Universal Robots PolyScope program: prod_v5.urp

Program prod_v5 (installation=prod directory=/home/ur/ursim-current/programs/programs.UR10 createdIn=3.14.1.1031110 lastSavedIn=3.14.1.1031110 robotSerialNumber=2018309999)
Calibrated DH parameters: a=[0.000066, -0.605508, -0.564633, 0.000003, 0.000034, 0]; d=[0.128223, 14.795741, 0.952357, -15.584568, 0.11573, 0.092195]; alpha=[1.569896, -0.006342, -0.005605, 1.571302, -1.571644, 0]; deltaTheta=[-0.000086, -0.153713, -0.001234, 0.154991, -0.000011, -0.000056]
InitVariablesNode variables(variable(name=last_task, expression=0), variable(name=print1, expression=False), variable(name=print2, expression=False), variable(name=print3, expression=False), variable(name=print_enable, expression=False), variable(name=vision_pos, expression=p[0,0,0,0,0,0]))
BeforeStart
  Script file /home/ur/ursim-current/programs/programs.UR10/readme.script
    | # SETUP INFO
    | # 1. Configure TCP
    | # 2. Calibrate vision planes A and B
    | # 3. Set the home position
    | # 4. Set variables at setup
    | 
    | # stack_ry - corresponds to tool rotation vector relative to stack
    | # print_width - width of the print label
    | # printer_width - width of the printer head
    | # ramp_distance - how far to reach constant speed
    | # clearance - how far away are we printing from the stack
    | # box_to_PA_XY - box coord to print area
    | # stack_a_to_ref, stack_b_to_ref - adjusts the vision plane calibration discrepancies
    | # TE_L2R - Task enum left to right
  Script file /home/ur/ursim-current/programs/programs.UR10/utils.script
    | def Max(a, b):
    |   if (a >= b):
    |     return a
    |   else:
    |     return b
    |   end
    | end
    | 
    | 
    | def Min(a, b):
    |   if (a <= b):
    |     return a
    |   else:
    |     return b
    |   end
    | end
  Folder Config
    'The tcp rotation components relative to stack'
    stack_ry := -180
    print_width := 0.04
    printer_width := 0.125
    ramp_dist := 0.05
    clearance := 0.04
    box_to_pa_XY := p[0.0325, -0.05, 0, 0, 0, 0]
    stack_a_to_ref := p[0, 0, 0, 0, 0, 0]
    stack_b_to_ref := p[0, 0, 0, 0, 0, 0]
    TE_L2R := 1
    TE_R2L := 2
  Folder Config Calcs
    print_range := (print_width+printer_width)/2
    runover := print_range+ramp_dist
  Folder Restart Checks
    tasks_equal := task≟current_task
    tasks_printing := task≠0 and current_task≠0 and print_enable
    resume_task := start_continue and tasks_equal and tasks_printing
    restart_task := GP_bool_in[3] and ( not resume_task) and tasks_printing
    print_enable := False
  Folder Keep current pos as home
    sp := get_actual_joint_positions()
    MoveJ speed 60 deg/s, acceleration 80 deg/s^2 (useActiveTCP=true)
      Waypoint Waypoint (Variable): variable=sp
  Folder Reset bits
    Set DigitalOutput pin=task_done; digitalValue=0
    Set DigitalOutput pin=task_active; digitalValue=0
    Set ExpressionOutput pin=current_task; expression=0
    Set DigitalOutput pin=homed; digitalValue=0
    Set DigitalOutput pin=moving_home; digitalValue=0
Robot Program (runOnlyOnce=false)
  If gantry_in_pos_a or gantry_in_pos_b
    If cancel_home
      Call PreTask
      Call MoveHome
    ElseIf task≟TE_L2R or task≟TE_R2L
      Call PreTask
      Call StartTask
      Call SetWaypoints
      Call MoveWaypoints
      Call FinishTask
SubProgram -> PreTask
SubProgram -> MoveHome
SubProgram -> StartTask
SubProgram -> SetWaypoints
SubProgram -> MoveWaypoints
SubProgram -> FinishTask
Thread Thread_1 (runOnlyOnce=false)
  'Monitors X position for printing'
  If print_enable
    vision_pos := pose_trans(pose_inv(reference), get_actual_tcp_pose())
    print1 := norm(vision_pos[0] - PA1[0]) ≤ print_range
    print2 := norm(vision_pos[0] - PA2[0]) ≤ print_range
    print3 := norm(vision_pos[0] - PA3[0]) ≤ print_range
  Set ExpressionOutput pin=printing; expression=(print1 or print2 or print3) and print_enable
  Script: sync()
SubProgram PreTask (keepSynchronizedWithDisk=false)
  If not (GP_bool_in[5] xor GP_bool_in[6])
    Popup Warning (haltProgram=false message=Err: Gantry not in pos inputType=Text)
  If gantry_in_pos_a
    reference := pose_add(stack_a, stack_a_to_ref)
  ElseIf gantry_in_pos_b
    reference := pose_add(stack_b, stack_b_to_ref)
  'Where is the miminimum Z relative to current pos'
  vision_pos_ex := pose_trans(pose_inv(reference), get_actual_tcp_pose())
  vision_pos_ex := pose_add(vision_pos_ex, p[0, 0, 2*clearance + GP_int_in[6]/1000 - vision_pos_ex[2], 0, 0, 0])
  CLEAR := pose_trans(reference, vision_pos_ex)
SubProgram MoveHome (keepSynchronizedWithDisk=false)
  Set ExpressionOutput pin=current_task; expression=0
  Set DigitalOutput pin=task_done; digitalValue=0
  Set DigitalOutput pin=task_active; digitalValue=0
  If not homed
    Set DigitalOutput pin=moving_home; digitalValue=1
    MoveL speed 100 mm/s, acceleration 100 mm/s^2 (useActiveTCP=true) feature=Base
      Waypoint home: motionParameters(blendRadius=0.05); TCP in base x=-358.527 y=-374.553 z=763.499 mm, rx=-0.681 ry=-1.6763 rz=1.7503 rad; joints [-9.825, -120.903, 126.278, -191.276, -37.611, 1.793] deg; flange x=-333.554 y=-184.862 z=721.81 mm, rx=-0.681 ry=-1.6763 rz=1.7503 rad
        Until REACHED_WAYPOINT (allowActions=true)
          Set DigitalOutput pin=homed; digitalValue=1
    Set DigitalOutput pin=moving_home; digitalValue=0
SubProgram StartTask (keepSynchronizedWithDisk=false)
  Set ExpressionOutput pin=current_task; expression=GP_int_in[0]
  Set DigitalOutput pin=task_active; digitalValue=1
SubProgram SetWaypoints (keepSynchronizedWithDisk=false)
  Folder Set Ordering
    B2 := p[X2/1000, Y/1000, Z/1000, 0, 0, 0]
    If current_task≟TE_L2R
      'Left to right (+ive)'
      xm := 1
      B1 := p[X1/1000, Y/1000, Z/1000, 0, 0, 0]
      B3 := p[X3/1000, Y/1000, Z/1000, 0, 0, 0]
    ElseIf current_task≟TE_R2L
      'Right to left (-ive)'
      xm := -1
      B1 := p[X3/1000, Y/1000, Z/1000, 0, 0, 0]
      B3 := p[X1/1000, Y/1000, Z/1000, 0, 0, 0]
  Folder Print Area Vars
    'Move the print areas relative to given box'
    'Do not overrwrite these'
    PA1 := pose_add(B1, box_to_pa_XY)
    PA2 := pose_add(B2, box_to_pa_XY)
    PA3 := pose_add(B3, box_to_pa_XY)
  Folder Calculate Waypoints
    PA1_EN := pose_add(PA1, p[-runover*xm, 0, clearance, 0, d2r(stack_ry), 0])
    PA3_EX := pose_add(PA3, p[+runover*xm, 0, clearance, 0, d2r(stack_ry), 0])
    APPROACH := pose_add(PA1_EN, p[0, 0, 2*clearance + GP_int_in[6]/1000 - PA1_EN[2], 0, 0, 0])
  Folder Reference Base
    PA1_EN := pose_trans(reference, PA1_EN)
    PA3_EX := pose_trans(reference, PA3_EX)
    APPROACH := pose_trans(reference, APPROACH)
SubProgram MoveWaypoints (keepSynchronizedWithDisk=false)
  'Minimum z position above entry'
  If homed
    MoveL speed 100 mm/s, acceleration 100 mm/s^2 (useActiveTCP=true) feature=Base
      Set ExpressionOutput pin=homed; expression=False
      Waypoint Waypoint (Variable): motionParameters(blendRadius=0.01); variable=APPROACH
        Until EXPRESSION (allowActions=false) ExpressionBranch=GP_bool_in[4]
      Waypoint Waypoint (Variable): motionParameters(blendRadius=0.01); variable=PA1_EN
        Until EXPRESSION (allowActions=false) ExpressionBranch=GP_bool_in[4]
  ElseIf resume_task
    'Resume from current position'
    Set ExpressionOutput pin=homed; expression=False
    resume_task := False
  ElseIf last_task≟TE_L2R and current_task≟TE_R2L and  not restart_task
    MoveL speed 100 mm/s, acceleration 100 mm/s^2 (useActiveTCP=true) feature=Base
      Set ExpressionOutput pin=homed; expression=False
      Waypoint Waypoint (Variable): motionParameters(blendRadius=0.01); variable=PA1_EN
        Until EXPRESSION (allowActions=false) ExpressionBranch=GP_bool_in[4]
  Else 
    restart_task := False
    MoveL speed 100 mm/s, acceleration 100 mm/s^2 (useActiveTCP=true) feature=Base
      Set ExpressionOutput pin=homed; expression=False
      Waypoint Waypoint (Variable): motionParameters(blendRadius=0.01); variable=CLEAR
        Until EXPRESSION (allowActions=false) ExpressionBranch=GP_bool_in[4]
      Waypoint Waypoint (Variable): motionParameters(blendRadius=0.01); variable=APPROACH
        Until EXPRESSION (allowActions=false) ExpressionBranch=GP_bool_in[4]
      Waypoint Waypoint (Variable): motionParameters(blendRadius=0.01); variable=PA1_EN
        Until EXPRESSION (allowActions=false) ExpressionBranch=GP_bool_in[4]
  'Move Across'
  MoveL speed 100 mm/s, acceleration 500 mm/s^2 (useActiveTCP=true) feature=Base
    print_enable := True
    Waypoint Waypoint (Variable): variable=PA3_EX
      Until EXPRESSION (allowActions=false) ExpressionBranch=GP_bool_in[4]
    print_enable := False
SubProgram FinishTask (keepSynchronizedWithDisk=false)
  'Acknowledgement sequence with PLC'
  last_task := current_task
  Set DigitalOutput pin=task_active; digitalValue=0
  Set DigitalOutput pin=task_done; digitalValue=1
  Wait Condition expression=task≟0 or cancel_home
  Set ExpressionOutput pin=current_task; expression=0
  Set DigitalOutput pin=task_done; digitalValue=0
